PROGRAM Safety_Manager
  VAR_EXTERNAL
    E_Stop : BOOL;
    Safety_OK : BOOL;
    System_Reset : BOOL;
  END_VAR

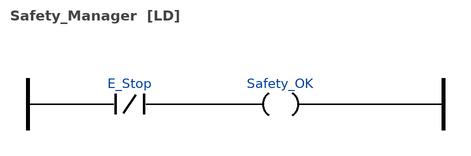
(* LD diagram, written out as Structured Text *)
Safety_OK := NOT E_Stop;
END_PROGRAM
